{attribute 'qualified_only'}
VAR_GLOBAL
	Parameters	: FB_Parameters_Store	:= (Pars := (
											Scale := 3.14,
											Etc := 42
										));
END_VAR

(* stored: Version 1.1.0.1, ProductVersion 3.1.4024.15
   GVL Parameters: Id {164fc1b2-9a73-4d71-8048-3d5a2e151eec} *)
